PROGRAM MAIN
VAR
END_VAR

POU();

END_PROGRAM

(* stored: Version 1.1.0.1, ProductVersion 3.1.4024.3
   POU MAIN: Id {aa289149-581f-420f-b1cc-f4b5e02d1d44}, SpecialFunc None *)
